// TwinCAT 3 PLC project PLC
// ProgramVersion: 3.1.4024.0
// libraries:
//   Tc2_Standard, * (Beckhoff Automation GmbH)
//   Tc2_System, * (Beckhoff Automation GmbH)
//   Tc3_Module, * (Beckhoff Automation GmbH)
// project tree:
//   / GlobalTextList.TcGTLO, PlcTask.TcTTO (not stored), VisualizationManager.TcVMO (not stored)
//   GVLs/ GVL.TcGVL
//   POUs/ FB_VisuSim.TcPOU (not stored), MAIN.TcPOU, FB_StateMachine.TcPOU (not stored)
//   VISUs/ Visu.TcVIS
// real-time tasks:
//   TASK PlcTask: cycle T#10ms, priority 20, ADS port 350
//   TASK VISU_TASK: cycle T#200000us, priority 30, ADS port 351

// ---- GVLs/GVL.TcGVL
(* -----------------------------------------------------------------------------
| This sample has been supplied by Beckhoff As-Is and is intended only as an   |
| example implementation. Functionality is not guaranteed.                     |
----------------------------------------------------------------------------- *)

{attribute 'qualified_only'}
VAR_GLOBAL
	// input
	bStart : BOOL;				// pulsante di start
	bStop : BOOL;				// pulsante di stop
	bBottle : BOOL;				// fotocellula FC1		

	// output
	bConveyor : BOOL;			// nastro trasportatore
	bWater : BOOL;				// riempimento acqua
	bMint : BOOL;				// riempimento menta	
	bCorking : BOOL;			// inserimento del tappo
END_VAR

// ---- POUs/MAIN.TcPOU
(* -----------------------------------------------------------------------------
| This sample has been supplied by Beckhoff As-Is and is intended only as an   |
| example implementation. Functionality is not guaranteed.                     |
----------------------------------------------------------------------------- *)

PROGRAM MAIN
VAR
	fbStateMachine : FB_StateMachine;
	fbVisuSim : FB_VisuSim;
END_VAR

(* -----------------------------------------------------------------------------
| This sample has been supplied by Beckhoff As-Is and is intended only as an   |
| example implementation. Functionality is not guaranteed.                     |
----------------------------------------------------------------------------- *)

fbStateMachine(
	bStart:= GVL.bStart, 
	bStop:= GVL.bStop, 
	bBottle:= GVL.bBottle,	 
);

GVL.bConveyor := fbStateMachine.bConveyor;
GVL.bWater := fbStateMachine.bWater;
GVL.bMint := fbStateMachine.bMint;	
GVL.bCorking := fbStateMachine.bCorking;

(* Visu and Simulation *)
fbVisuSim(bConveyor:= GVL.bConveyor);
GVL.bBottle := fbVisuSim.bBottle;

END_PROGRAM

// ---- GlobalTextList.TcGTLO
TEXTLIST GlobalTextList
  663 = '%s'
  445 = 'START'
  530 = 'STOP'
END_TEXTLIST

// ---- VISUs/Visu.TcVIS
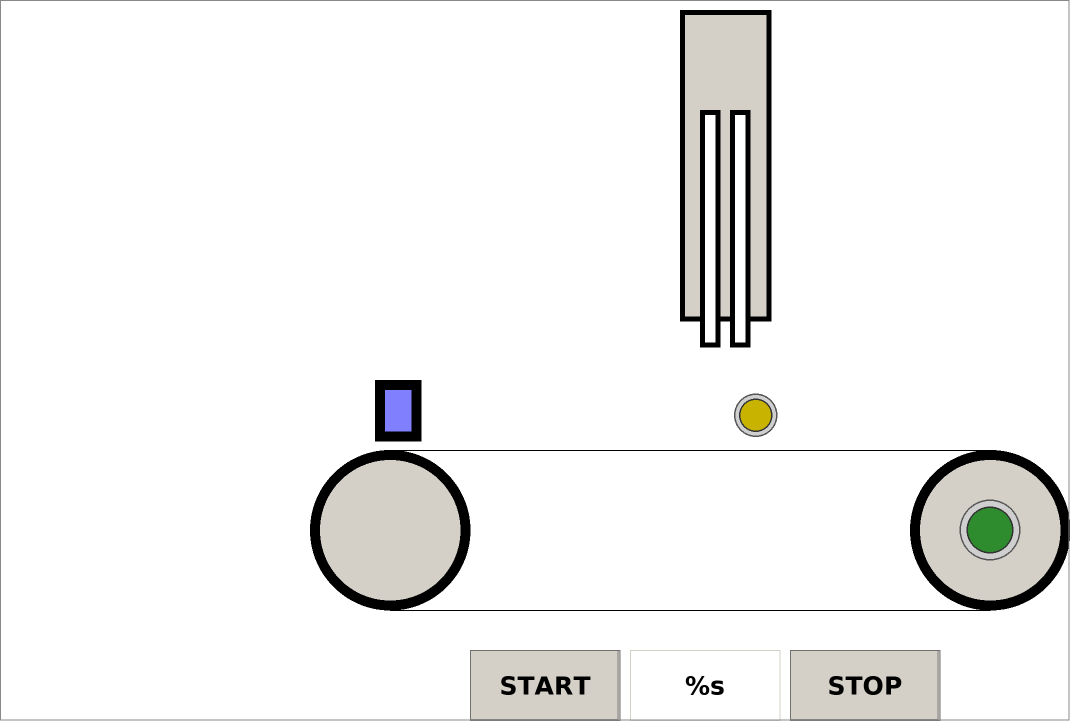
VISUALIZATION Visu  // 1070x721
    Rectangle (680,10 91x311), colour toggle: GVL.bCorking
        p2738717112: (TO_REAL(GVL.bCorking) * 50.0)
    Ellipse (310,450 160x160)
    Line (390,450) (990,450)
    Ellipse (910,450 160x160)
    Line (390,610) (990,610)
    Lamp1 (955,495 70x70), variable: GVL.bConveyor, style: Lamp-Lamp1-Green
    Rectangle (700,110 20x237), colour toggle: GVL.bWater
    Rectangle (730,110 20x237), colour toggle: GVL.bMint
    Button (470,650 150x71), "START"
        tap GVL.bStart
    Button (790,650 150x71), "STOP"
        tap GVL.bStop
    Textfield (630,650 150x71), "%s", text variable: MAIN.fbStateMachine.nStep
    Lamp1 (730,390 51x50), variable: GVL.bBottle, style: Lamp-Lamp1-Yellow
    RoundedRectangle (375,380 46x61)
        p3560616238: MAIN.fbVisuSim.fPos * 5.0
END_VISUALIZATION
